// TIA Portal project "babu_exhaustfanAndstove" (V15)

(* hardware
DEVICE "S7-1200 station_1"  S7-1200 Station
   slot 0: "Rack_0"  S7-1200 Rack  Rack  V1.0
   slot 1: "PLC_1"  CPU 1212C DC/DC/DC  6ES7 212-1AE40-0XB0  V4.2
*)

// ===== PLC "PLC_1"  CPU 1212C DC/DC/DC =====

VAR_GLOBAL   // PLC tag table "Tag table_1"
   "STOVE" AT %M0.0 : Bool;
   "MEMORY" AT %M0.1 : Bool;
   "FAN" AT %Q0.2 : Bool;
   "SWITCH" AT %Q0.3 : Bool;
   "S1" AT %Q0.4 : Bool;
   "STOVE1" AT %Q0.5 : Bool;
   "FAN1" AT %Q0.6 : Bool;
END_VAR

// folder: System blocks/Program resources

DATA_BLOCK "IEC_Timer_0_DB"   // DB1
{ S7_Optimized_Access := 'TRUE' }
AUTHOR : Simatic
FAMILY : IEC
NAME : IEC_TMR
VERSION : 1.0
// stored: InstanceOfName IEC_TIMER
"IEC_TIMER"
BEGIN
END_DATA_BLOCK

DATA_BLOCK "IEC_Timer_0_DB_2"   // DB3
{ S7_Optimized_Access := 'TRUE' }
AUTHOR : Simatic
FAMILY : IEC
NAME : IEC_TMR
VERSION : 1.0
// stored: InstanceOfName IEC_TIMER
"IEC_TIMER"
BEGIN
END_DATA_BLOCK

// folder: (top level)

ORGANIZATION_BLOCK "Main"   // OB1, LAD, ProgramCycle
TITLE = "Main Program Sweep (Cycle)"
{ S7_Optimized_Access := 'TRUE' }
VERSION : 0.1
   VAR_INPUT
      Initial_Call : Bool;   // Initial call of this OB
      Remanence : Bool;   // =True, if remanent data are available
   END_VAR
BEGIN

REGION Network 1
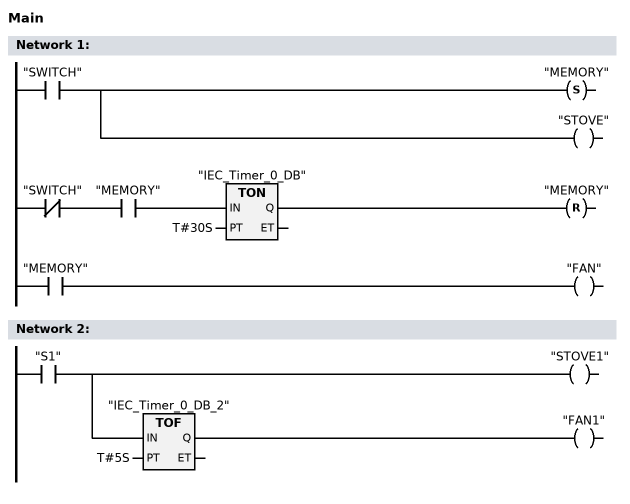
   IF "SWITCH" THEN "MEMORY" := TRUE; END_IF;
   "STOVE" := "SWITCH";
   "IEC_Timer_0_DB".TON(IN := NOT "SWITCH" AND "MEMORY", PT := T#30S);
   IF "IEC_Timer_0_DB".Q THEN "MEMORY" := FALSE; END_IF;
   "FAN" := "MEMORY";
END_REGION

REGION Network 2
   "STOVE1" := "S1";
   "IEC_Timer_0_DB_2".TOF(IN := "S1", PT := T#5S);
   "FAN1" := "IEC_Timer_0_DB_2".Q;
END_REGION
END_ORGANIZATION_BLOCK